FUNCTION_BLOCK Pulse2
VAR_INPUT
	button1: BOOL;
	time_fuction: INT;
END_VAR
VAR_OUTPUT
	Flag: BOOL;
END_VAR
VAR
	Timer1: TON;
END_VAR

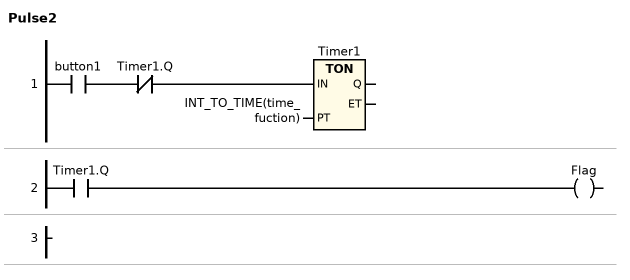
// NETWORK 1
Timer1(IN := button1 AND NOT Timer1.Q, PT := INT_TO_TIME(time_fuction)); // TON

// NETWORK 2
Flag := Timer1.Q;

// NETWORK 3

END_FUNCTION_BLOCK

(* stored: Version 1.1.0.1, ProductVersion 3.1.4024.12
   POU Pulse2: Id {a7a31bf4-497f-42db-ace3-2461a43ac371}, SpecialFunc None *)
